FUNCTION_BLOCK FB_AUT_110 EXTENDS FB_AUT_ABSTRACT
(****************************************************************************)
(*	POU_AUT_zxx			Bausteinaufrufe Station	zxx							*)
(*	Status				ungetestet											*)
(*  Version:			1.0													*)
(*	Beschrieb:																*)
(*																			*)
(*	Abläufe:			FB_ABLzxxA		Hauptablauf							*)
(*																			*)
(*																			*)
(* 	25.09.2019/Dj															*)
(****************************************************************************)
(*	dd.mm.yyyy   KZ    x.y			Beschrieb								*)
(****************************************************************************)
VAR_INPUT
    (* spezifische Eingänge *)

END_VAR
VAR_OUTPUT
    (* spezifische Ausgänge *)

END_VAR
VAR
    (* Bausteine *)
    fb_Pnp    : FB_ABL_110_Pnp;
    fb_Feeder : FB_ABL_110_Feeder;

END_VAR

VAR CONSTANT
    ROT_TABLE_FREE_MAX_Y : REAL := 200.0; // If Y and Z axis is more than this value, the feeder cannot move
    ROT_TABLE_FREE_MAX_Z : REAL := 200.0; // If Z and Y axis is more than this value, the feeder cannot move
END_VAR

(*******************************************************************)
(* Timer *)
(*******************************************************************)

(*******************************************************************)
(* Flanken / Merker *)
(*******************************************************************)
//MANU CYCLE
IF (enIN_State = StateMANU) AND xIN_ManuCycle THEN
    xManuCycle := TRUE;
END_IF;

IF (enIN_State <> StateMANU) OR xOUT_Done THEN
    xManuCycle := FALSE;
END_IF

//NEXT STEP
xNextStep := (enIN_State > StateSTEP) OR
             ((enIN_State = StateSTEP) AND xIN_Step) OR
             ((enIN_State = StateMANU) AND xManuCycle);

//RESET
xReset := (enIN_State < StateREADY) AND (enIN_State <> StateINIT) AND NOT xManuCycle;

(*******************************************************************)
(* Bausteinaufrufe Abläufe *)
(*******************************************************************)

fb_Pnp(xIN_Reset          := xReset,
       xIN_Init           := xIN_Init,
       xIN_Quit           := xIN_Quit,
       xIN_Start          := enIN_State = enState.StateAUTO, //AND _FB_ABL_100A.xOUT_Done AND _FB_ABL_100A.xOUT_Ready,
       xIN_Sperre         := NOT xIN_On,
       xIN_NextStep       := xNextStep,
       xIN_AlarmAktiv     := xIN_AlarmAktiv,
       xIN_DryCycle       := xIN_DryCycle,
       xIN_RestartCYCL    := enIN_State = enState.StateAUTO, // only restart when the mover has move out
       enIN_State         := enIN_State,
       tIN_Timeout        := tIN_Timeout,
       pxFG_Freigabe      := ADR(xDummy),
       Mover              := THIS^.Mover,
       xIN_PceReadyToPick := fb_Feeder.xOUT_Done);

fb_Feeder(xIN_Reset       := xReset,
          xIN_Init        := xIN_Init,
          xIN_Quit        := xIN_Quit,
          xIN_Start       := enIN_State = enState.StateAUTO, //AND _FB_ABL_100A.xOUT_Done AND _FB_ABL_100A.xOUT_Ready, 
          xIN_Sperre      := NOT xIN_On,
          xIN_NextStep    := xNextStep,
          xIN_AlarmAktiv  := xIN_AlarmAktiv,
          xIN_DryCycle    := xIN_DryCycle,
          xIN_RestartCYCL := enIN_State = enState.StateAUTO, // only restart when the mover has move out
          enIN_State      := enIN_State,
          tIN_Timeout     := tIN_Timeout,
          pxFG_Freigabe   := ADR(xDummy),
          // special
          xIN_PickPiece            := fb_Pnp.xOUT_PickPiece,
          xIN_RotTableBlockedByPnp := (ST110_Axis.axis110_01Y.rActPos > ROT_TABLE_FREE_MAX_Y) AND
                                      (ST110_Axis.axis110_02Z.rActPos > ROT_TABLE_FREE_MAX_Z));

(*******************************************************************)
(* Mover reset flags *)
(*******************************************************************)

(*******************************************************************)
(* OUTPUT *)
(*******************************************************************)
xOUT_InitDone := fb_Pnp.xOUT_InitDone AND fb_Feeder.xOUT_InitDone;
xOUT_Ready    := fb_Pnp.xOUT_Ready AND fb_Feeder.xOUT_Ready;
xOUT_Done     := fb_Pnp.xOUT_Done;
xOUT_ErrFlag  := fb_Pnp.xOUT_ErrFlag;
xOUT_Wait     := fb_Pnp.xOUT_Wait;
xOUT_AlarmST  := xOUT_ErrFlag;

(*******************************************************************)
(* Bausteinaufruf Error Station *)
(*******************************************************************)
// POU_ERR_VORLAGE(xIN_QUIT:=xIN_Quit , pstrArIN_ALARM:=ADR(HMI.strArALARM[1]));

METHOD GiveMover : IProcessSampleMover
VAR_INPUT
	mover : REFERENCE TO FB_Mover;
END_VAR
IF __ISVALIDREF(mover) THEN
    THIS^.Mover                       REF= mover;
END_IF
END_METHOD

(* % of completion of the process *)
PROPERTY iCompletionPC : INT
GET
iCompletionPC := THIS^.fb_Pnp.iOUT_ProcessCompletion;
END_GET
END_PROPERTY

PROPERTY ProcessExecution : ProcessExecution_e
GET
ProcessExecution := THIS^._ProcessExecution;
END_GET
SET
THIS^._ProcessExecution := ProcessExecution;
END_SET
END_PROPERTY

METHOD TakeMover : IProcessSampleMover
VAR_INPUT
END_VAR
THIS^.Mover REF= 0;
END_METHOD

PROPERTY xBusy : BOOL
GET
xBusy := THIS^.fb_Pnp.xOUT_Busy;
END_GET
SET
END_SET
END_PROPERTY

PROPERTY xDone : BOOL
GET
xDone := THIS^.fb_Pnp.xOUT_Ready OR THIS^.fb_Pnp.xOUT_Done;
END_GET
END_PROPERTY

PROPERTY xMoverPathFree : BOOL
GET
xMoverPathFree := THIS^.fb_Pnp.xOUT_MoverFree OR THIS^.fb_Pnp.xOUT_Ready OR THIS^.fb_Pnp.xOUT_Done;
END_GET
END_PROPERTY

PROPERTY xMoverShouldLeave : BOOL
GET
xMoverShouldLeave := THIS^.fb_Pnp.iOUT_Step = ST110_Pnp_e.SYNC_MOVER_LEAVE;
END_GET
END_PROPERTY

END_FUNCTION_BLOCK

(* stored: Version 1.1.0.1, ProductVersion 3.1.4024.6
   POU FB_AUT_110: Id {3a75638e-4197-4ed4-a9b7-03c2fb32897f}, SpecialFunc None
   Method GiveMover: Id {90505fb1-9a4c-45d5-b06e-16a18772176e}
   Property iCompletionPC: Id {f03aab34-0709-45b8-80fe-12aa7c735bba}
   Get Get: Id {c855a333-89d4-4129-bf32-6b480d79436f}
   Property ProcessExecution: Id {9944028e-71e4-4f6c-ab9d-2e450d36f1e7}
   Get Get: Id {e439908e-0dcd-4313-9915-d6f50d6a1e3c}
   Set Set: Id {72e06213-981e-443b-b6c4-73d8e8052a5d}
   Method TakeMover: Id {d84cb916-2f66-4d9a-b351-183c45d9b25f}
   Property xBusy: Id {a5e462d0-5361-4950-a5f3-f24e71556501}
   Get Get: Id {3ea2fb3d-7ff1-4760-b35f-20e1f7d0a75a}
   Set Set: Id {06ec9da9-7624-4525-8133-0d040f619b4c}
   Property xDone: Id {6724bbc4-60f1-4aa1-85a4-8236f2174d20}
   Get Get: Id {059441f4-0e47-47a7-add9-12f3a94a07c1}
   Property xMoverPathFree: Id {597cbc1b-58ec-44cf-8369-e55c696d7510}
   Get Get: Id {48ce9e58-a174-4804-944b-d3b0235f1954}
   Property xMoverShouldLeave: Id {97a4c977-4d48-474e-8d38-73231615f1f2}
   Get Get: Id {2040f511-ef63-4808-9c4b-0956653d64fb} *)
